DATA_BLOCK "HMISystemDB"
VAR
  DisplayRows : Int;
  MaxPage : Int;
  Rows : Int;
  UnEnableGroup : Bool;
  DisplaySymbol : Bool;
  "DisplaySymbol Time" : Int;
  SymbolText : Array[1..4] of Int;
  HMICylinderBypass : Array[1..50] of Struct;
  HMI_Axis : "HMI_Axis";
END_VAR
BEGIN
END_DATA_BLOCK
